Universal Robots PolyScope program: old.urp

Program old (installation=remote_weld directory=/programs/usbdisk/new folder_1 createdIn=3.1.17195.0 lastSavedIn=5.12.2.1101534 robotSerialNumber=20225202267)
Calibrated DH parameters: a=[0.000057, -0.560337, -0.56987, 0.000044, 0.000023, 0]; d=[0.180974, -304.223407, 295.067386, 9.330269, 0.119831, 0.115671]; alpha=[1.570416, 0.000812, 0.004616, 1.569457, -1.570316, 0]; deltaTheta=[0, -0.415128, 6.624286, 0.074029, 0.000002, -0.000001]
BeforeStart
  open := socket_open("192.168.0.56",50000)
  Loop While (checkContinuously=false) expression=open≟ False
    open := socket_open("192.168.0.56",50000)
  targetPos := p[0,0,0,0,0,0]
  counter := 6
  Start_code := [0,0]
  act_current := 0
  act_voltage := 0
  act_wirefeeder := 0
Robot Program (runOnlyOnce=false)
  Loop Forever
    If Start_code[1]==1
      URCap WeldItem (Migapath, Smooth Robotics ApS)
        URCap Weld seam (Migapath, Smooth Robotics ApS) dataModel(titleKey=Weld seam, dataModelVersion=1, programVersion=1)
          URCap AirPoint (Migapath, Smooth Robotics ApS) dataModel(title_key=Airpoint, jump_visible=true, pose_has_been_offset=false, move_key=MOVEJ, Pose(key=move_pose_key, Position(key=posePosition, Length(key=X value=0.481824 unit=M), Length(key=Y value=-0.817952 unit=M), Length(key=Z value=0.368197 unit=M)), Rotation(key=poseRotation, Angle(key=RX value=-1.7397 unit=RAD), Angle(key=RY value=1.830526 unit=RAD), Angle(key=RZ value=0.698368 unit=RAD))), JointPositions(key=move_joint_key, JointPosition(key=[1], Angle(key=pos value=-0.838325 unit=RAD)), JointPosition(key=[2], Angle(key=pos value=-1.984976 unit=RAD)), JointPosition(key=[3], Angle(key=pos value=-0.845022 unit=RAD)), JointPosition(key=[4], Angle(key=pos value=-1.848216 unit=RAD)), JointPosition(key=[5], Angle(key=pos value=1.554361 unit=RAD)), JointPosition(key=[6], Angle(key=pos value=0.749368 unit=RAD))))
          URCap AirPoint (Migapath, Smooth Robotics ApS) dataModel(title_key=Airpoint_1, pose_has_been_offset=false, movel_speed_key=40.0, move_key=MOVEL, Pose(key=move_pose_key, Position(key=posePosition, Length(key=X value=0.72217 unit=M), Length(key=Y value=-0.616582 unit=M), Length(key=Z value=0.144361 unit=M)), Rotation(key=poseRotation, Angle(key=RX value=-1.60381 unit=RAD), Angle(key=RY value=1.72815 unit=RAD), Angle(key=RZ value=0.875332 unit=RAD))), JointPositions(key=move_joint_key, JointPosition(key=[1], Angle(key=pos value=-0.585806 unit=RAD)), JointPosition(key=[2], Angle(key=pos value=-2.101727 unit=RAD)), JointPosition(key=[3], Angle(key=pos value=-1.048484 unit=RAD)), JointPosition(key=[4], Angle(key=pos value=-1.669571 unit=RAD)), JointPosition(key=[5], Angle(key=pos value=1.689211 unit=RAD)), JointPosition(key=[6], Angle(key=pos value=1.004684 unit=RAD))))
          URCap AirPoint (Migapath, Smooth Robotics ApS) dataModel(title_key=Startpoint, move_key=MOVEL, movel_speed_key=20.0, pose_has_been_offset=false, Pose(key=move_pose_key, Position(key=posePosition, Length(key=X value=0.590252 unit=M), Length(key=Y value=-0.552083 unit=M), Length(key=Z value=0.098623 unit=M)), Rotation(key=poseRotation, Angle(key=RX value=-1.702594 unit=RAD), Angle(key=RY value=1.653046 unit=RAD), Angle(key=RZ value=0.860692 unit=RAD))), JointPositions(key=move_joint_key, JointPosition(key=[1], Angle(key=pos value=-0.611194 unit=RAD)), JointPosition(key=[2], Angle(key=pos value=-1.836078 unit=RAD)), JointPosition(key=[3], Angle(key=pos value=-1.509732 unit=RAD)), JointPosition(key=[4], Angle(key=pos value=-1.440839 unit=RAD)), JointPosition(key=[5], Angle(key=pos value=1.690846 unit=RAD)), JointPosition(key=[6], Angle(key=pos value=0.896729 unit=RAD))))
          SuppressedNode
            Script: socket_send_int(3)
          SuppressedNode
            Wait Condition expression=Start_code[1]==2
          URCap Arc On (Migaweld, Smooth Robotics ApS) dataModel(arcOnWaitTime=0.0)
          URCap Paths: (Migapath, Smooth Robotics ApS)
            URCap Welding path (Migapath, Smooth Robotics ApS) dataModel(titleKey=Linear_1, selectedPathType=Linear, selectedPattern=None, end_has_been_offset=false, Pose(key=endPose, Position(key=posePosition, Length(key=X value=0.562124 unit=M), Length(key=Y value=-0.551211 unit=M), Length(key=Z value=0.100844 unit=M)), Rotation(key=poseRotation, Angle(key=RX value=-1.649017 unit=RAD), Angle(key=RY value=1.677805 unit=RAD), Angle(key=RZ value=0.860658 unit=RAD))), JointPositions(key=endJoint, JointPosition(key=[1], Angle(key=pos value=-0.637368 unit=RAD)), JointPosition(key=[2], Angle(key=pos value=-1.815933 unit=RAD)), JointPosition(key=[3], Angle(key=pos value=-1.53044 unit=RAD)), JointPosition(key=[4], Angle(key=pos value=-1.455311 unit=RAD)), JointPosition(key=[5], Angle(key=pos value=1.69991 unit=RAD)), JointPosition(key=[6], Angle(key=pos value=0.912258 unit=RAD))))
          URCap Arc Off (Migaweld, Smooth Robotics ApS) dataModel(arcOffWaitTime=0.5)
          Script: socket_send_int(4)
          URCap AirPoint (Migapath, Smooth Robotics ApS) dataModel(title_key=Airpoint, pose_has_been_offset=false, move_key=MOVEL, Pose(key=move_pose_key, Position(key=posePosition, Length(key=X value=0.577963 unit=M), Length(key=Y value=-0.645486 unit=M), Length(key=Z value=0.188127 unit=M)), Rotation(key=poseRotation, Angle(key=RX value=-1.68074 unit=RAD), Angle(key=RY value=1.854334 unit=RAD), Angle(key=RZ value=0.57428 unit=RAD))), JointPositions(key=move_joint_key, JointPosition(key=[1], Angle(key=pos value=-0.626149 unit=RAD)), JointPosition(key=[2], Angle(key=pos value=-1.736851 unit=RAD)), JointPosition(key=[3], Angle(key=pos value=-1.507974 unit=RAD)), JointPosition(key=[4], Angle(key=pos value=-1.364844 unit=RAD)), JointPosition(key=[5], Angle(key=pos value=1.562636 unit=RAD)), JointPosition(key=[6], Angle(key=pos value=1.041202 unit=RAD))))
Thread Thread_1 (runOnlyOnce=false)
  Script: act_current=read_input_integer_register(7)
  SuppressedNode
    Script: act_current=15
  Script: act_voltage=read_input_integer_register(6)
  Script: act_wirefeeder=read_input_integer_register(7)
  Start_code := socket_read_ascii_float(1)
  If Start_code[1]==2 (checkContinuously=true)
    Folder Value
      Current := str_cat(to_str(act_current),",")
      Voltage := str_cat(to_str(act_voltage),",")
    Script: socket_send_string(str_cat(str_cat(Current,Voltage),to_str(act_wirefeeder)))
  Wait Sleep waitTime=0.1
